(* CoDeSys 2.3.9.41 project: MO_752.pro *)
(* Libraries: STANDARD.LIB 4.10.05 11:14:46, IECSFC.LIB 13.4.06 15:51:28, SYSLIBTIME.LIB 20.2.06 13:31:16, SYSTASKINFO.LIB 20.2.06 13:31:38, ANALYZATION.LIB 5.10.99 09:05:06, arm7_specific.lib 12.5.10 15:26:52, ComService.lib 21.5.09 14:28:28, Ind_Mode.lib 26.8.10 18:05:16, ModBus.lib 27.5.09 09:22:38, Sound.lib 17.10.08 11:37:02, SysLibCom.lib 20.2.06 13:31:08, Util.lib 18.5.10 15:14:28 *)

(* PLC configuration (modules and I/O channels)
PLC73 [Root] node -1, in %IB0 out %QB0 {BName = #NМеню ПЛК73#A0; MinCycleLenght = 1; MaxCycleLenght = 1000}
  Configuration [ID10050] node 0, in %IB0 out %QB0 {BName = #NКонфигурация#A0}
    DInputs [ID10051] node 0, in %IB0.0 out %QB0.0 {BName = #NДискретные Вх.#A0}
      AT %IB0.0.0 [DInput] Битовая маска входов {CPString128 = #NСост.Дискр.Вх.#Fr.Cn#H2D26#A3#T02#O#B0120#V2; DinLM = #NЛогика Дискр.Вх#Finv.D#H62C2#A0#T02#D00#MFF#B0121#V2; DinFl = #NПост.Ф.ДребКонт#FTin.F#HF89F#A0#U0017#T02#D0A#MFF#B0122}
    Outputs [ID10057] node 1, in %IB0.1 out %QB0.1 {BName = #NВУ#A0}
      AT %QD0.1.0 [AnalogOutput0] Выход 1 {CPString128 = #NСост.ВУ1#Fr.oe#HE894#I00#A0#T00#C3#M+1.00E+00#O#B0000; AoutPWMP = #NПериод ШИМ ВУ1#Fthpd#H7BFE#I00#A0#U0017#T01#D03E8#MFDE8#L0002#B0123; AoutPWMM = #NМин.имп.ШИМ ВУ1#Ft.L#I00#B012B#A0#U0017#T01#D0032#L0001#M1388; AoutSafeValue = #NБезоп.сост.ВУ1#FO.ALr#I00#B0010#A0#C3#T00#D+0.00E+00#M+1.00E+00}
      AT %QD0.1.1 [AnalogOutput1] Выход 2 {CPString128 = #NСост.ВУ2#Fr.oe#I01#B0002#A0#O#C3#T00#M+1.00E+00; AoutPWMP = #NПериод ШИМ ВУ2#Fthpd#I01#B0124#A0#U0017#T01#D03E8#L0002#MFDE8; AoutPWMM = #NМин.имп.ШИМ ВУ2#Ft.L#I01#B012C#A0#U0017#T01#D0032#L0001#M1388; AoutSafeValue = #NБезоп.сост.ВУ2#FO.ALr#I01#B0012#A0#C3#T00#D+0.00E+00#M+1.00E+00}
      AT %QD0.1.2 [AnalogOutput2] Выход 3 {CPString128 = #NСост.ВУ3#Fr.oe#I02#B0004#A0#O#C3#T00#M+1.00E+00; AoutPWMP = #NПериод ШИМ ВУ3#Fthpd#I02#B0125#A0#U0017#T01#D03E8#L0002#MFDE8; AoutPWMM = #NМин.имп.ШИМ ВУ3#Ft.L#I02#B012D#A0#U0017#T01#D0032#L0001#M1388; AoutSafeValue = #NБезоп.сост.ВУ3#FO.ALr#I02#B0014#A0#C3#T00#D+0.00E+00#M+1.00E+00}
      AT %QD0.1.3 [AnalogOutput3] Выход 4 {CPString128 = #NСост.ВУ4#Fr.oe#HE894#I03#A0#T00#C3#M+1.00E+00#O#B0006; AoutPWMP = #NПериод ШИМ ВУ4#Fthpd#I03#B0126#A0#U0017#T01#D03E8#L0002#MFDE8; AoutPWMM = #NМин.имп.ШИМ ВУ4#Ft.L#I03#B012E#A0#U0017#T01#D0032#L0001#M1388; AoutSafeValue = #NБезоп.сост.ВУ4#FO.ALr#I03#B0016#A0#C3#T00#D+0.00E+00#M+1.00E+00}
      AT %QD0.1.4 [AnalogOutput4] Выход 5 {CPString128 = #NСост.ВУ5#Fr.oe#HE894#I04#A0#T00#C3#M+1.00E+00#O#B0008; AoutPWMP = #NПериод ШИМ ВУ5#Fthpd#I04#B0127#A0#U0017#T01#D03E8#L0002#MFDE8; AoutPWMM = #NМин.имп.ШИМ ВУ5#Ft.L#I04#B012F#A0#U0017#T01#D0032#L0001#M1388; AoutSafeValue = #NБезоп.сост.ВУ5#FO.ALr#I04#B0018#A0#C3#T00#D+0.00E+00#M+1.00E+00}
      AT %QD0.1.5 [AnalogOutput5] Выход 6 {CPString128 = #NСост.ВУ6#Fr.oe#HE894#I05#A0#T00#C3#M+1.00E+00#O#B000A; AoutPWMP = #NПериод ШИМ ВУ6#Fthpd#I05#B0128#A0#U0017#T01#D03E8#L0002#MFDE8; AoutPWMM = #NМин.имп.ШИМ ВУ6#Ft.L#I05#A0#B0130#U0017#T01#D0032#L0001#M1388; AoutSafeValue = #NБезоп.сост.ВУ6#FO.ALr#I05#B001A#A0#C3#T00#D+0.00E+00#M+1.00E+00}
      AT %QD0.1.6 [AnalogOutput6] Выход 7 {CPString128 = #NСост.ВУ7#Fr.oe#I06#B000C#A0#O#C3#T00#M+1.00E+00; AoutPWMP = #NПериод ШИМ ВУ7#Fthpd#I06#B0129#A0#U0017#T01#D03E8#L0002#MFDE8; AoutPWMM = #NМин.имп.ШИМ ВУ7#Ft.L#I06#B0131#A0#U0017#T01#D0032#L0001#M1388; AoutSafeValue = #NБезоп.сост.ВУ7#FO.ALr#I06#B001C#A0#C3#T00#D+0.00E+00#M+1.00E+00}
      AT %QD0.1.7 [AnalogOutput7] Выход 8 {CPString128 = #NСост.ВУ8#Fr.oe#I07#B000E#A0#O#C3#T00#M+1.00E+00; AoutPWMP = #NПериод ШИМ ВУ8#Fthpd#I07#B012A#A0#U0017#T01#D03E8#L0002#MFDE8; AoutPWMM = #NМин.имп.ШИМ ВУ8#Ft.L#I07#A0#B0132#U0017#T01#D0032#L0001#M1388; AoutSafeValue = #NБезоп.сост.ВУ8#FO.ALr#I07#B001E#A0#C3#T00#D+0.00E+00#M+1.00E+00}
    AInputs [ID10055] node 2, in %IB0.2 out %QB0.2 {BName = #NАналоговые Вх.#A0; Spay = #NКоррекция ХС#Fcj-.c#B0133#A0#U002A#T03#D01}
      AT %ID0.2.0 [AnalogInput0] Аналоговый вход 1 {CPString128 = #NВход 1#Fread#H8784#I00#A3#T10#C2#O#B0020#V3; AinType = #NТип датчика 1#Fin-t#H932D#I00#A0#U002F#T04#D01#M15#B0134; InFD = #NПост. фильтра 1#Fin.Fd#I00#B013C#A0#U0018#T01#D0005#M0708; InFG = #NПолоса Фильтра1#Fin.FG#I00#B0030#A0#T00#D+1.00E+01#L+0.00E+01#M+9.99E+03}
      AT %ID0.2.1 [AnalogInputTime0] Время измерения 1
      AT %ID0.2.2 [AnalogInput1] Аналоговый вход 2 {CPString128 = #NВход 2#Fread#H8784#I01#A3#T10#C2#O#B0022#V3; AinType = #NТип датчика 2#Fin-t#H932D#I01#A0#U002F#T04#D01#M15#B0135; InFD = #NПост. фильтра 2#Fin.Fd#I01#B013D#A0#U0018#T01#D0005#M0708; InFG = #NПолоса Фильтра2#Fin.FG#I01#B0032#A0#T00#D+1.00E+01#L+0.00E+01#M+9.99E+03}
      AT %ID0.2.3 [AnalogInputTime1] Время измерения 2
      AT %ID0.2.4 [AnalogInput2] Аналоговый вход 3 {CPString128 = #NВход 3#Fread#H8784#I02#A3#T10#C2#O#B0024#V3; AinType = #NТип датчика 3#Fin-t#I02#B0136#A0#U002F#T04#D01#M15; InFD = #NПост. фильтра 3#Fin.Fd#I02#B013E#A0#U0018#T01#D0005#M0708; InFG = #NПолоса Фильтра3#Fin.FG#I02#B0034#A0#T00#D+1.00E+01#L+0.00E+01#M+9.99E+03}
      AT %ID0.2.5 [AnalogInputTime2] Время измерения 3
      AT %ID0.2.6 [AnalogInput3] Аналоговый вход 4 {CPString128 = #NВход 4#Fread#H8784#I03#A3#T10#C2#O#B0026#V3; AinType = #NТип датчика 4#Fin-t#I03#B0137#A0#U002F#T04#D01#M15; InFD = #NПост. фильтра 4#Fin.Fd#I03#B013F#A0#U0018#T01#D0005#M0708; InFG = #NПолоса Фильтра4#Fin.FG#I03#A0#B0036#T00#D+1.00E+01#L+0.00E+01#M+9.99E+03}
      AT %ID0.2.7 [AnalogInputTime3] Время измерения 4
      AT %ID0.2.8 [AnalogInput4] Аналоговый вход 5 {CPString128 = #NВход 5#Fread#I04#B0028#C2#A3#O#V3#T10; AinType = #NТип датчика 5#Fin-t#I04#B0138#A0#U002F#T04#D01#M15; InFD = #NПост. фильтра 5#Fin.Fd#I04#B0140#A0#U0018#T01#D0005#M0708; InFG = #NПолоса Фильтра5#Fin.FG#I04#B0038#A0#T00#D+1.00E+01#L+0.00E+01#M+9.99E+03}
      AT %ID0.2.9 [AnalogInputTime4] Время измерения 5
      AT %ID0.2.10 [AnalogInput5] Аналоговый вход 6 {CPString128 = #NВход 6#Fread#I05#B002A#C2#A3#O#V3#T10; AinType = #NТип датчика 6#Fin-t#I05#B0139#A0#U002F#T04#D01#M15; InFD = #NПост. фильтра 6#Fin.Fd#I05#B0141#A0#U0018#T01#D0005#M0708; InFG = #NПолоса Фильтра6#Fin.FG#I05#B003A#A0#T00#D+1.00E+01#L+0.00E+01#M+9.99E+03}
      AT %ID0.2.11 [AnalogInputTime5] Время измерения 6
      AT %ID0.2.12 [AnalogInput6] Аналоговый вход 7 {CPString128 = #NВход 7#Fread#I06#B002C#C2#A3#O#V3#T10; AinType = #NТип датчика 7#Fin-t#I06#B013A#A0#U002F#T04#D01#M15; InFD = #NПост. фильтра 7#Fin.Fd#I06#B0142#A0#U0018#T01#D0005#M0708; InFG = #NПолоса Фильтра7#Fin.FG#I06#B003C#A0#T00#D+1.00E+01#L+0.00E+01#M+9.99E+03}
      AT %ID0.2.13 [AnalogInputTime6] Время измерения 7
      AT %ID0.2.14 [AnalogInput7] Аналоговый вход 8 {CPString128 = #NВход 8#Fread#H8784#I07#A3#T10#C2#O#B002E#V3; AinType = #NТип датчика 8#Fin-t#I07#B013B#A0#U002F#T04#D01#M15; InFD = #NПост. фильтра 8#Fin.Fd#I07#B0143#A0#U0018#T01#D0005#M0708; InFG = #NПолоса Фильтра8#Fin.FG#I07#B003E#A0#T00#D+1.00E+01#L+0.00E+01#M+9.99E+03}
      AT %ID0.2.15 [AnalogInputTime7] Время измерения 8
    MR1_Outputs [ID10053] node 3, in %IB0.3 out %QB0.3 {BName = #NВУ МР1#A0}
      AT %QB0.3.0 [DOutput] ВУ МР1 {CPString128 = #NСост.ВУ МР1#Fr.oe.s#HA9F4#A0#T02#O#B0144#V2}
    Additional [ID10059] node 4, in %IB0.4 out %QB0.4 {BName = #NДоп.пар-ры#A0}
      AT %QB0.4.0 [LCDLight] Подсветка {CPString128 = #NЯрк.подсв.ЖКИ#Find.i#H1845#A0#T02#D2D#M32#B0145}
      AT %QB0.4.1 [LCDContrast] Контраст {CPString128 = #NКонтраст ЖКИ#Find.C#B0146#A0#T02#D19#L05#M20}
      AT %IW0.4.2 [KBD] Клавиатура {CPString128 = #NСост.клавиатуры#Fkbrd#B0147#A3#O#T02; KBDBeep = #NЗвук кнопок#Fbeep#B0148#A0#U002A#T03#D01}
      AT %QD0.4.3 [RTS] Часы контроллера {RTSPar = #NВремя и дата#FrtC#HFA30#A0#T05#O#B0040}
      AT %QB0.4.4 [LED] Светодиоды {CPString128 = #NСос.светодиодов#Find.L#HF304#A0#T02#D00#M3F#L00#O#B0149#V2}
    Versions [ID10060] node 5, in %IB0.5 out %QB0.5 {BName = #NВерсииПрошивок#A0}
      AT %QB0.5.0 [DevName] Имя устройства {CPString128 = #NИмя устройства#Fdev#B0042#A3#O#T08}
      AT %IB0.5.1 [HardVer] Прошивка {CPString128 = #NВерсия прошивки#Fver#B004A#A3#O#T08}
      AT %QB0.5.2 [SoftVer] Программа {CPString128 = #NВерсияПрограммы#Fp.ver#B0052#A3#O#T08}
    RS-1 [ID10061] node 6, in %IB0.6 out %QB0.6 {BName = #NНастр.RS-1#A0; RSBPS = #NСкорость#FbPS#I00#B014A#A0#U0046#T04#D00#M09; RSWLen = #NДлина слова#FLen#I00#B014B#A0#U0005#T04#D03#M03; RSPrt = #NЧётность#Fprty#I00#B014C#A0#U009A#T04#D04#M04; RSStp = #NСтоп биты#Fsbit#I00#B014D#A0#U00A1#T04#D00#M02; RSALen = #NДлина адреса#Fa.len#I00#B014E#A0#U0055#T03#D00; RSAdr = #NАдрес прибора#FAddr#I00#B014F#A0#T01#D0010#M07FF; RSDl = #NЗадержка ответа#FRs.dl#I00#B0150#A0#U0017#T02#D05#M32}
    RS-2 [ID10062] node 7, in %IB0.7 out %QB0.7 {BName = #NНастр.RS-2#A0; RSBPS = #NСкорость#FbPS#I01#B0151#A0#U0046#T04#D00#M09; RSWLen = #NДлина слова#FLen#I01#B0152#A0#U0005#T04#D03#M03; RSPrt = #NЧётность#Fprty#I01#B0153#A0#U009A#T04#D04#M04; RSStp = #NСтоп биты#Fsbit#I01#B0154#A0#U00A1#T04#D00#M02; RSALen = #NДлина адреса#Fa.len#I01#B0155#A0#U0055#T03#D00; RSAdr = #NАдрес прибора#FAddr#I01#B0156#A0#T01#D0010#M07FF; RSDl = #NЗадержка ответа#FRs.dl#I01#B0157#A0#U0017#T02#D05#M32}
  WorkInd [ID10100] node 1, in %IB1 out %QB1 {WIChanelCount = 6}
  SubMenu [ID11000] node 2, in %IB2 out %QB2 {BName = #NВетка#A0}
  SubMenu [ID11000] node 3, in %IB3 out %QB3 {BName = #NВетка#A0}
  SubMenu [ID11000] node 4, in %IB4 out %QB4 {BName = #NВетка#A0}
*)

(* Global variable list: Global_Variables *)
VAR_GLOBAL CONSTANT

	byMU110Address: BYTE:=11;				(*адрес МУ-110*)
	byMV110Address: BYTE:=22;				(*адрес МВ-110*)

END_VAR
VAR_GLOBAL
	bDInput1 AT %IX0.0.0.0: BOOL;
	bDInput2 AT %IX0.0.0.1: BOOL;
	bDInput3 AT %IX0.0.0.2: BOOL;
	bDInput4 AT %IX0.0.0.3: BOOL;
	bDInput5 AT %IX0.0.0.4: BOOL;
	bDInput6 AT %IX0.0.0.5: BOOL;
	bDInput7 AT %IX0.0.0.6: BOOL;
	bDInput8 AT %IX0.0.0.7: BOOL;

	rOutput1 AT %QD0.1.0: REAL;
	rOutput2 AT %QD0.1.1: REAL;
	rOutput3 AT %QD0.1.2: REAL;
	rOutput4 AT %QD0.1.3: REAL;
	rOutput5 AT %QD0.1.4: REAL;
	rOutput6 AT %QD0.1.5: REAL;
	rOutput7 AT %QD0.1.6: REAL;
	rOutput8 AT %QD0.1.7: REAL;

	rAInput1 AT %ID0.2.0: REAL;
	rAInput2 AT %ID0.2.2: REAL;
	rAInput3 AT %ID0.2.4: REAL;
	rAInput4 AT %ID0.2.6: REAL;
	rAInput5 AT %ID0.2.8: REAL;
	rAInput6 AT %ID0.2.10: REAL;
	rAInput7 AT %ID0.2.12: REAL;
	rAInput8 AT %ID0.2.14: REAL;

	kbrd AT %IW0.4.2: WORD;
	led  AT %QB0.4.4: BYTE;
	n: WORD := 0;
END_VAR
VAR_GLOBAL RETAIN
	wFilterTimeRet: 	WORD	:= 3000;    (*время фильтра поплавка в мс*)
	tempMaxRet: 		BYTE	:= 95;		(*максим. температура*)
	timeMaxRet: 		WORD	:= 999;		(*максим. время*)
	USDelayRet: 		WORD	:= 0;		(*время блокировки повторного включения УЗ в сек*)
	hystRet: 			WORD	:= 2;		(*гистерезис *10^(-2) гр.С*)
	pumpModeRet: 	    BOOL;				(*режим работы насоса (TRUE - работает постоянно, FALSE - с заданной частотой и скважностью*)
	pumpTimeLo:         WORD;				(*массив для задания времени бездействия насоса в минутах*)
	pumpTimeHi: 		WORD;				(*массив для задания продолжительности работы насоса в секундах*)
	APRet: 		        ARRAY [US_1..Wash] OF APST;				(*параметры автоматической программы*)
	powerOffDelayRet: 	WORD	:= 15;		(*задержка отключения питания генераторов в секундах*)
	genOnDelayRet: 	    WORD	:= 500;		(*время между включениями генераторов в мс*)
    fillDelay:          WORD    := 5;       (*задержка закрытия электроклапана наполнения воды*)
    ventTime:           WORD    := 0;       (*задержка гидролока*)
	timePump:			WORD    := 1;
	temp_Air:			WORD;
	time_dry:			WORD;
END_VAR

(* Global variable list: GVL_APBool *)
VAR_GLOBAL CONSTANT
    WarmWait :BYTE:=0;    (*отложенный старт*)
    DynContr :BYTE:=1;    (*динамическое управление*)
    RotOn    :BYTE:=2;    (*качание*)
END_VAR

(* Global variable list: GVL_CONST *)
VAR_GLOBAL CONSTANT
	iQtyD7Line: 		INT		:=25;		(*количество строк в расписании недельного таймера*)
	iMaxSelScrParam: 	INT		:=26;		(*максимальное количество строк на экране выбора параметра*)
	iStQty: 			INT		:=10;		(*количество шагов автоматической программы*)
	tUSDelay: 			TIME	:=t#1m;		(*задержка повторной подачи питания на УЗГ*)
	GlobalMaxRand: 		USINT	:=18;		(*количество рандомных значений и максимальное значение рандома*)
END_VAR

(* Data type in BathFB *)
TYPE APST :
STRUCT
	areSt:		ARRAY [1..iStQty] OF StAPE;        (*массив шагов автоматической программы*)
	arwTime:	ARRAY [1..iStQty] OF WORD;         (*временной параметр шага в минутах*)
	byTemp:		BYTE;                              (*заданная температура*)
	byBool:		BYTE;                              (*состояние программных ключей. Описываются в GVL_APBoolE*)
	byTempAir:	BYTE;
END_STRUCT
END_TYPE

(* Data type *)
TYPE Button :
STRUCT
    pusk:            ARRAY [US_1..Wash] OF BOOL;   (*Пуск*)
    stop:            ARRAY [US_1..Wash] OF BOOL;   (*Стоп*)
    emStop:          BOOL;   (*Аварийный стоп*)
	pusk_dry:		BOOL;
	stop_dry:		BOOL;
    puskDrain:       BOOL;   (*Пуск слива*)
    puskFill:        BOOL;   (*Пуск наполнения*)
    puskPump:        BOOL;   (*Пуск насоса*)
    puskBubbles:     BOOL;   (*Пуск барботажа*)
	warmOn:          BOOL;
END_STRUCT
END_TYPE

(* Data type in BathFB *)
TYPE ButtonBath :
STRUCT
	Pusk:          BOOL;   (*Пуск цикла*)
	PuskDrain:     BOOL;   (*Пуск слива*)
	PuskFill:      BOOL;   (*Пуск наполнения*)
	PuskPump:      BOOL;   (*Пуск насоса*)
	PuskBubbles:   BOOL;   (*Пуск барботажа*)
	Stop:          BOOL;   (*Стоп*)
	StopDrain:     BOOL;   (*Стоп слива*)
	StopFill:      BOOL;   (*Стоп наполнения*)
	emStop:        BOOL;   (*Аварийная остановка*)
END_STRUCT
END_TYPE

(* Data type in BathFB *)
TYPE ButtonEvent :
STRUCT
   (* кнопка нажата, устанавливается на один цикл *)
   downEvent:    BOOL;

   (* нажатие дольше секунды *)
   longPush:     BOOL;

   (* число, на которое надо инкрементировать, сначала 1,
   начиная с 3 секунды увеличиваеться на 1 каждую секунду *) 
   incr:         BYTE;
END_STRUCT
END_TYPE

(* Data type *)
TYPE Control :
STRUCT
	heatUSTank:		BOOL;                    (*нагрев в баке УЗВ*)
	heatWashTank:	BOOL;                    (*нагрев в баке ополаскивания*)
	pump:			BOOL;                    (*насосы*)
	lampAtt:		BOOL;                    (*лампа "Внимание"*)
	warning_bath:	ARRAY [US_1..Wash] OF BOOL;
	warning_dry:	BOOL;
	lampWork:		BOOL;                    (*лампа "Работа"*)
	lamp_work_dry:	BOOL;
	lamp_work_bath:	ARRAY [US_1..US_2] OF BOOL;
	lampTopLevel:	BOOL;                    (*лампа "Верхняя группа УЗГ"*)
	lampLowerLevel:	BOOL;                    (*лампа "Нижняя группа УЗГ"*)
	genPower:		BOOL;                    (*питание генераторов*)
	skim:			BOOL;                    (*скиммеры*)
	gener:			ARRAY [1..36] OF BOOL;   (*генераторы*)
	heat_air:		BOOL;
	fan:			BOOL;
END_STRUCT
END_TYPE

(* Data type in BathFB *)
TYPE ControlBath :
STRUCT
   us:                  BOOL;      (*ультразвук*)
   warmBath:            BOOL;      (*нагрев ванны*)
   warmTank:            BOOL;      (*нагрев бака*)
   rotFo:               BOOL;      (*вращение вперед*)
   rotRe:               BOOL;      (*вращение назад*)
   ventBfromNet:        BOOL;      (*вентиль из сети*)
   pumpBfromTank:       BOOL;      (*фильтрационный насос*)
   ventBPocketToNet:    BOOL;      (*вентиль из кармана в сеть*)
   ventBPocketToTank:   BOOL;      (*вентиль из кармана в бак*)
   ventBToNet:          BOOL;      (*вентиль из ванны в сеть*)
   ventBToTank:         BOOL;      (*вентиль из ванны в бак*)
   ventBarb:            BOOL;      (*барботаж*)
   skim:                BOOL;      (*скиммер*)
   dry:                 BOOL;      (*сушка*)
   dryFan:              BOOL;      (*вентилятор сушки*)
END_STRUCT
END_TYPE

(* Data type in D7Timer *)
TYPE D7TLineST :    (*структура одной линии расписания 7дн таймера*)
STRUCT
    wTimeOfWeek:    WORD;    (*время недели в минутах, к этому времени надо нагреть*)
    byTemp:         BYTE;    (*поддерживаемая температура*)
    byDur:          BYTE;    (*продолжительность в часах*)
END_STRUCT
END_TYPE

(* Data type in D7Timer *)
TYPE DoWE :
(
    Mon:=0,
    Tue,
    Wed,
    Thu,
    Fri,
    Sat,
    Sun
);
END_TYPE

(* Data type in BathFB *)
(*Дополнительные выходы ванны*)
TYPE ExtOutST :
STRUCT
    remTime:     TIME;    (*оставшееся время*)
    bathEmpty:   BOOL;    (*ванна пуста*)
END_STRUCT
END_TYPE

(* Data type in BathFB *)
(*дополнительные параметры ванны*)
TYPE ExtParamST :
STRUCT
    (*Нагреватели*)
    heatPlace:        HeatPlaceE;    (*место расположения нагревателя*)
    heaterInTank:     BOOL;          (*расположение ТЭН в баке*)
    deltaHyst:        WORD;          (*гистерезис нагрева (e(-2))*)
    waitTemp:         BYTE;          (*температура режима ожидания (с недельного таймера или заданная вручную)*)
    mixTimeHi:        WORD;          (*время работы перемешивания в секундах*)
    mixTimeLo:        WORD;          (*время ожидания перемешивания в минутах*)
    pumpTimeHi:       WORD;          (*работа насоса в секундах*)
    pumpTimeLo:       WORD;          (*ожидание насоса в минутах*)
    mixStart:         BOOL;          (*время между включениями барботажа при нагреве в минутах*)
    mixDur:           WORD;          (*время барботажа при нагреве в секундах*)

    (*Вентили*)
    ventTime:         WORD;          (*время работы вентиля в секундах*)
    drainDelay:       WORD;          (*дополнительное время слива в секундах*)
    fillDelay:        WORD;          (*дополнтельное время наполнения в секундах*)
    pumpDelay:        WORD;          (*дополнительное время насоса в секундах*)
    fillTankDelay:    WORD;          (*дополнительное время наполнения бака в секундах*)
    dontDrain:        BOOL;          (*не сливать ванну*)

    (*барабан*)
    rotTime:          WORD;          (*период качания в миллисекундах*)
    rotDur:           WORD;          (*продолжительность качания в секундах*)
    rotSlack:         WORD;          (*продолжительность бездействия в секундах*)
    filtrRot:         BOOL;          (*вращение при фильтрации*)

    (*скиммер*)
    skimTimeHi:       WORD;          (*время работы скиммера в минутах*)
    skimTimeLo:       WORD;          (*время ожидания скиммера в минутах*)

END_STRUCT
END_TYPE

(* Data type in BathFB *)
TYPE FlE :
(
    NoFl,    (*нет жидкости*)
    TMS,
    water
);
END_TYPE

(* Data type in BathFB *)
(*расположение нагревателя*)
TYPE HeatPlaceE :
(
    US_1,
    US_2,
    Wash
);
END_TYPE

(* Data type in Other *)
TYPE kbrd_tip :
(
    off:=0,
    DOWN:=4,
    UP:=8,
    ENTER:=16,
    OUT:=64,
    ALT:=128,
    F1:=1,
    F2:=2,
    F3:=256,
    pusk_stop:=32,
    ALT_F1:=129,
    ALT_F3:=384
);
END_TYPE

(* Data type *)
TYPE Level :
(
    BathTop,
    BathMiddle,
    BathLower,
    TankTop,
    TankMiddle,
    TankLower,
    USBlock,
    USBlockTop,
    WarmBlock,
    PumpBlock,
    BarbBlock,
    SkimerBlock,
    FillBathStop
);
END_TYPE

(* Data type in BathFB *)
TYPE LevelBath :
STRUCT
    BathTop:        BOOL;       (*Верхний уровень в ванне*)
    BathMiddle:     BOOL;       (*Средний уровень в ванне*)
    BathLower:      BOOL;       (*Нижний уровень в ванне*)
    TankTop:        BOOL;       (*Верхний уровень в баке*)
    TankMiddle:     BOOL;       (*Средний уровень в баке*)
    TankLower:      BOOL;       (*Нижний уровень в баке*)
    USBlock:        BOOL;       (*Уровень блокировки уровня ультразвука*)
    USBlockTop:     BOOL;       (*Уровень блокировки верхнего уровня ультразвука*)
    WarmBlock:      BOOL;       (*Уровень блокировки нагрева*)
    PumpBlock:      BOOL;       (*Уровень блокировки насоса*)
    BarbBlock:      BOOL;       (*Уровень блокировки барботажа*)
    SkimerBlock:    BOOL;       (*Уровень блокировки скимера*)
    FillBathStop:   BOOL;       (*Уровень заполнения*)
END_STRUCT
END_TYPE

(* Data type *)
TYPE MBStepE :
(
    StepSelect,
    MV110Read,
    MU110Write
);
END_TYPE

(* Data type *)
TYPE ModuleAddr :
(
    A2 := 22,
    A3 := 33,
    A4 := 44,
    A5 := 55,
    A6 := 66,
    A7 := 77
);
END_TYPE

(* Data type *)
TYPE Screens :
(
	s_info,

	s_osnovnoy_US_1,
	s_osnovnoy_US_2,
	s_osnovnoy_Wash,
	s_osnovnoy_Dry,

	s_nastroyki,
	s_nastroyki_ext,

	s_time,
	s_time_us_1,
	s_time_us_2,
	s_time_dry,

	s_tem,
	s_tem_us_1,
	s_tem_us_2,
	s_tem_wash,
	s_tem_dry,

	s_tMaxSet,
	s_temHSet
);
END_TYPE

(* Data type in Other *)
TYPE SelectScreenAddStruc :
STRUCT
    strIn: STRING(5);    (*строка, дописываемая между ВЫХОД и ВХОД*)
END_STRUCT
END_TYPE

(* Data type *)
TYPE Sensor :
STRUCT
    level:			ARRAY [BathTop..FillBathStop, US_1..Wash] OF BOOL;	(*массив уровней*)
    button:			Button;									(*кнопки*)
    genState:		ARRAY [1..36] OF BOOL;					(*состояние генераторов*)
    tempBath:		ARRAY [US_1..Wash] OF REAL;				(*температура ванны*)
    overloadPump:	BOOL;									(*Перегрев насоса*)
	temAir:			REAL;
	cover:			BOOL;
END_STRUCT
END_TYPE

(* Data type in BathFB *)
TYPE SensorBath :
STRUCT
    level:			LevelBath;   (*Уровни*)
    tempBath:		REAL;        (*Температура ванны*)
    tempTank:		REAL;        (*Температура бака*)
	tempAir:		REAL;
	button:			ButtonBath;  (*Кнопки*)
    Fl:				FlE;         (*тип жидкости в ванне*)
    warmOn:			BOOL;        (*нагрев включен*)
    mixOn:			BOOL;        (*перемешивание включен*)
    pause:			BOOL;        (*Пауза АП*)
    rotOn:			BOOL;        (*Включение вращения*)
    flReset:		BOOL;        (*Сброс типа жидкости*)
	overloadPump:	BOOL;        (*перегрузка насоса*)
END_STRUCT
END_TYPE

(* Data type in Other *)
(*дополнительные настройки для блока экрана установки параметра*)
TYPE SetScreenAddStruc :
STRUCT
    Extend:        BOOL;                        (*разрешает работу блока в режиме задания разных велечин*)
    in_var:        ARRAY[1..3] OF DWORD;        (*задаваемая переменная*)
    in_var_min:    ARRAY[1..3] OF  DWORD;       (*мин значение задаваемой переменной*)
    in_var_max:    ARRAY[1..3] OF  DWORD;       (*макс значение задаваемой переменной*)
    UnitParam:     ARRAY[1..3] OF  STRING(16);  (*в каких единицах ведется задание минуты секунды градусы и тд*)
    EnableF3:      BOOL;                        (*разрешить третью единицу измерения*)
    bDoWSet:       BOOL;                        (*задаваемый параметр - день недели*)
    iValInc:       INT;                         (*шаг увеличения величины*)
END_STRUCT
END_TYPE

(* Data type in Other *)
TYPE StAPE:
(
    Wait:=0,
    WarmTank,
    WarmBath,
    FillFromTank,
    US,
    FiltrToTank,
    DrainToTank,
    FillFromNet,
    US2,
    FiltrToNet,
    DrainToNet,
    FillTank,
    ManToNet,
    ManToTank,
    Skip,
    Barb,
    Barb_and_Filtr,
    Dry,
    DeGas,
    Warning,
    Pump,
	Cooling,
	Heating
);
END_TYPE

(* Data type in BathFB *)
TYPE StE :
(
    on,
    off1,
    not_enabled
);
END_TYPE

(* Data type *)
TYPE VarST :
STRUCT
    pby:      POINTER TO BYTE;
    type_:    VarType;
END_STRUCT
END_TYPE

(* Data type *)
TYPE VarType :
(
    BYTE_,
    WORD_,
    DWORD_,
    REAL_,
    DINT_,
    DWORD_30,
    DWORD_500
);
END_TYPE

(* POU PLC_PRG, ST *)
PROGRAM PLC_PRG
VAR
	bInit:              BOOL;
	warning:            BOOL;
	C:                  INT;
	D:                  BOOL;

	encoder_:			Encoder;
	TON50ms:            TON;

	bath:               ARRAY [US_1..Wash] OF BFBv4;                           (*массив ФБ ванн*)
	block:              ARRAY [US_1..Wash] OF BlockFBv2;                       (*блокировки*)
	sens:               Sensor;                          (*структура датчиков*)
	contr:              Control;                         (*структура управления*)
	filtr:              digitalFiltr;
	buttons:            KeyboardFB;
	variable:           VarST;
	HYST_Air:			HYST;
	TON_heat_air:		TON;
	TON_fan:			TON;
	TONP:				TONP;
	start_heat_air:		BOOL;
	stape:				StAPE;

	(*modbus*)
	bOpenPort:          BOOL        := 0;
	ePorts:             PORTS       := 0;
	stSettings:         COMSETTINGS;
	oComService:        COM_SERVICE;
	arMBuffer:          ARRAY [0..255] OF BYTE;
	tTimeOut:           TIME        := t#100ms;      (*время таймаута порта*)
	eMBStep:            MBStepE     := MV110Read;  (*кейс модбаса*)
	udErr:              UDINT       :=0;            (*счетчик ошибок*)
	wBuffer:            WORD;

	mbA2:               WORD;
	arTON:              ARRAY [1..2] OF TON;

	oMB_16:             MB_WR_REGS;                 (*функция Modbus 16*)
	oMB_03:             MB_RD_HOLD_REGS;            (*функция Modbus 03*)
	oMB_06:				MB_WR_SNG_REG;				(*запись значения в один регистр хранения (Preset Single Register).*)

	TONMBDelay:         TON;                        (*таймер задержки modbus*)
	tMBDelay:           TIME        := t#10ms;     (*задержка modbus*)
	bMBStepSelect:      BOOL;                       (*выбор запись/чтение*)

	(*indicator*)
	Current_screen:     screens     := s_info;
	TONInfo:            TON;
	str:                ARRAY [1..4] OF STRING(16);
	pred_str:           ARRAY [1..4] OF STRING(16);
	SelectScreen:       SelectScreenFB;
	SetScreen:          SetScreenFB;

END_VAR
VAR_TEMP

	I:                  INT;
	k:                  INT;
	j:                  INT;
	iStTmp:             INT;                        (*шаг АП*)
	line:               INT;                        (*строка индикатора*)

END_VAR
IF NOT(bInit) THEN
    acInit();									(*инициализация*)
ELSE

	buttons(kbrd := kbrd);
	acMB();
	SelectScreen.encoder_(A := bDInput6, B := bDInput5, button := bDInput7, connected := TRUE);
	SetScreen.pSelect := ADR(SelectScreen);
	C := SelectScreen.encoder_.counter;
	D := SelectScreen.encoder_.press;

	encoder_(A := bDInput6, B := bDInput5, button := bDInput7, connected := TRUE);


	(*назначение входов*)
	sens.tempBath[US_1]			:= rAInput1;
	sens.tempBath[US_2]			:= rAInput2;
	sens.tempBath[Wash]			:= rAInput3;
	sens.temAir					:= rAInput4;

	sens.button.emStop			:= bDInput1;

	sens.level[BathLower, US_1]	:= mbA2.0;
	sens.level[BathLower, US_2]	:= mbA2.1;
	sens.level[BathLower, Wash]	:= mbA2.2;
	sens.button.pusk[US_1]		:= mbA2.4;
	sens.button.stop[US_1]		:= mbA2.5;
	sens.button.pusk[US_2]		:= mbA2.6;
	sens.button.stop[US_2]		:= mbA2.7;
	sens.button.pusk_dry		:= mbA2.8;
	(*sens.button.stop_dry		:= mbA2.9;*)

	(*назначение входов ванн*)
	FOR i := US_1 TO Wash DO
		bath[i].sens.button.Pusk               := sens.button.pusk[i];
		bath[i].sens.button.Stop               := sens.button.stop[i] ;
		bath[i].sens.pause                     := NOT sens.level[BathLower, i];
		bath[i].sens.tempBath                  := sens.tempBath[i];
		bath[i].sens.level.BathLower           := sens.level[BathLower, i];
		bath[i].sens.warmOn                    := TRUE;
		bath[i].param.heaterInTank             := TRUE;
		bath[i].param.deltaHyst                := hystRet;
		bath[i].sens.button.emStop             := sens.button.emStop;
		bath[i].sens.level.USBlock := bath[i].sens.level.WarmBlock := bath[i].sens.level.BathLower;
	END_FOR


	FOR i := US_1 TO Wash DO
		bath[i](stAP:=APRet[i]);
		block[i]();
	END_FOR

	(*управление*)
	CASE stape OF
		Wait:
			contr.heat_air	:= FALSE;
			contr.fan		:= FALSE;
			IF sens.button.pusk_dry AND (temp_Air <> 0) AND (time_dry <> 0) THEN
				stape := Heating;
			END_IF
		Heating:
			contr.heat_air := HYST_Air.nagrev;
			contr.fan := TRUE;
			IF sens.temAir >= temp_Air THEN
				stape:= Dry;
			END_IF
			IF sens.button.stop_dry THEN
				contr.heat_air := FALSE;
				stape := Cooling;
			END_IF
		Dry:
			contr.heat_air := HYST_Air.nagrev;
			contr.fan := TRUE;
			TONP(P := FALSE, IN := TRUE, PT := TO_MIN(time_dry));
			IF TONP.Q OR sens.button.stop_dry THEN
				contr.heat_air := FALSE;
				TONP(IN:= FALSE);
				stape := Cooling;
			END_IF
		Cooling:
			TON_fan(IN := TRUE, PT := TO_MIN(5));
			IF TON_fan.Q THEN
				TON_fan(IN:= FALSE);
				stape := Wait;
			END_IF
	END_CASE

	HYST_Air.temperatura := temp_Air;
	HYST_Air(ENABLE := stape = Dry OR stape = Heating, temInput := sens.temAir	, temperaturaH := hystRet);

	FOR i := US_1 TO Wash DO
		contr.warning_bath[i]	:= NOT bath[i].sens.level.BathLower OR bath[i].sens.button.emStop OR (bath[i].sens.tempBath < 0);
	END_FOR
	contr.warning_dry			:= sens.temAir < 0;



	contr.lamp_work_bath[US_1]	:= bath[US_1].eStAP <> Wait;
	contr.lamp_work_bath[US_2]	:= bath[US_2].eStAP <> Wait;
	contr.lamp_work_dry			:= stape <> Wait;
	contr.lampAtt				:= contr.warning_bath[US_1] OR contr.warning_bath[US_2] OR contr.warning_bath[Wash] OR contr.warning_dry;

	(*Назначение выходов*)
	rOutput3 := BOOL_TO_REAL(contr.lampAtt);
	rOutput1 := BOOL_TO_REAL(contr.lamp_work_bath[US_1] OR contr.lamp_work_bath[US_2] OR contr.lamp_work_dry);

	rOutput5 := BOOL_TO_REAL(contr.lamp_work_bath[US_1]);
	rOutput6 := BOOL_TO_REAL(contr.lamp_work_bath[US_2]);
	rOutput7 := BOOL_TO_REAL(contr.lamp_work_dry);

	led.0 := contr.warning_bath[US_1];
	led.1 := contr.warning_bath[US_2];
	led.2 := contr.warning_bath[Wash];
	led.3 := contr.warning_dry;

	(*вызов действия индикации*)
	TON50ms(IN:=TRUE,PT:=t#50ms);
	IF TON50ms.Q THEN
		TON50ms(IN:=FALSE);
		acIndicator();
	END_IF
END_IF
END_PROGRAM
ACTION acIndicator:
CASE Current_screen OF

	s_info:

		Switch_To_Single_Mode();				(*переход в монопольный режим*)
		str[1] := '      ООО       ';
		str[2] := 'Александра-Плюс ';
		str[3] := '                ';
		str[4] := '     МО-752     ';
		TONInfo(IN := TRUE, PT := t#5s);
		IF TONInfo.Q THEN
			TONInfo(IN := FALSE);
			encoder_(reset := TRUE);
			Current_screen := s_osnovnoy_US_1;
		END_IF

	s_osnovnoy_US_1:
		encoder_(reset := FALSE);
		SelectScreen(kbrd := kbrd, QtyParam := 3);
		line := 1;
		str[line] := ' МО-752    УЗВ1 ';
		line := 2;
		IF bath[US_1].eStAP <> Wait THEN
			str[line] := CONCAT('Время     ', TIME_TO_MMSS(bath[US_1].extOutB.remTime));
		ELSE
			str[line] := CONCAT('Время     ', TIME_TO_MMSS(TO_MIN(APRet[US_1].arwTime[2])));
		END_IF

		line := 3;
		str[line] := CONCAT('Нагрев ', TEMP_TO_STRING(bath[US_1].sens.tempBath));
		str[line] := CONCAT(str[line], '/');
		str[line] := CONCAT(str[line], DWORD_TO_STRING (APRet[US_1].byTemp ));
		str[line] := CONCAT(str[line], '$9BС');
		line := 4;
		IF sens.tempBath[US_1] < 0 THEN
			str[line] := ' неисправно ТС  ';
			warning :=TRUE;
		ELSIF sens.button.emStop  THEN
			str[line] := ' Авар. останов! ';
			warning :=TRUE;
		ELSIF NOT bath[US_1].sens.level.BathLower  THEN
			str[line] := 'низкий ур. р-ра ';
			warning :=TRUE;
		ELSIF stape = Heating THEN
			str[line] := '    подогрев    ';
			warning :=FALSE;
		ELSIF stape = Dry THEN
			str[line] := '     сушка      ';
			warning :=FALSE;
		ELSIF bath[US_1].eStAP = US THEN
			str[line] := '   ультразвук   ';
			warning :=FALSE;
		ELSIF stape = Cooling THEN
			str[line] := '   охлаждение   ';
			warning :=FALSE;
		ELSIF bath[US_1].eStAP = Wait THEN
			str[line] := 'ожидание старта ';
			warning :=FALSE;
		END_IF
		IF SelectScreen.encoder_.press AND SelectScreen.encoder_.enable OR SelectScreen.kbrd = F1 THEN
			SelectScreen.encoder_(enable := FALSE);
			Current_screen := s_nastroyki;
		END_IF
		IF SelectScreen.kbrd = ALT_F3 THEN
			Current_screen := s_nastroyki_ext;
		END_IF

		IF (encoder_.counter >= 1) THEN
			Current_screen := s_osnovnoy_US_2;
			encoder_(reset := TRUE);
		ELSIF encoder_.counter < 0 THEN
			encoder_(reset := TRUE);
		END_IF


	s_osnovnoy_US_2:
		encoder_(reset := FALSE);
		SelectScreen(kbrd := kbrd, QtyParam := 3);
		line := 1;
		str[line] := ' МО-752    УЗВ2 ';
		line := 2;
		IF bath[US_2].eStAP <> Wait THEN
			str[line] := CONCAT('Время     ', TIME_TO_MMSS(bath[US_2].extOutB.remTime));
		ELSE
			str[line] := CONCAT('Время     ', TIME_TO_MMSS(TO_MIN(APRet[US_2].arwTime[2])));
		END_IF

		line := 3;
		str[line] := CONCAT('Нагрев ', TEMP_TO_STRING(bath[US_2].sens.tempBath));
		str[line] := CONCAT(str[line], '/');
		str[line] := CONCAT(str[line], DWORD_TO_STRING (APRet[US_2].byTemp ));
		str[line] := CONCAT(str[line], '$9BС');
		line := 4;
		IF sens.tempBath[US_2] < 0 THEN
			str[line] := ' неисправно ТС  ';
			warning :=TRUE;
		ELSIF sens.button.emStop  THEN
			str[line] := ' Авар. останов! ';
			warning :=TRUE;
		ELSIF NOT bath[US_2].sens.level.BathLower  THEN
			str[line] := 'низкий ур. р-ра ';
			warning :=TRUE;
		ELSIF stape = Heating THEN
			str[line] := '    подогрев    ';
			warning :=FALSE;
		ELSIF stape = Dry THEN
			str[line] := '     сушка      ';
			warning :=FALSE;
		ELSIF bath[US_2].eStAP = US THEN
			str[line] := '   ультразвук   ';
			warning :=FALSE;
		ELSIF stape = Cooling THEN
			str[line] := '   охлаждение   ';
			warning :=FALSE;
		ELSIF bath[US_2].eStAP = Wait THEN
			str[line] := 'ожидание старта ';
			warning :=FALSE;
		END_IF
		IF SelectScreen.encoder_.press AND SelectScreen.encoder_.enable OR SelectScreen.kbrd = F1 THEN
			SelectScreen.encoder_(enable := FALSE);
			Current_screen := s_nastroyki;
		END_IF
		IF SelectScreen.kbrd = ALT_F3 THEN
			Current_screen := s_nastroyki_ext;
		END_IF
		IF (encoder_.counter <= - 1) THEN
			Current_screen := s_osnovnoy_US_1;
			encoder_(reset := TRUE);
		ELSIF (encoder_.counter >= 1) THEN
			Current_screen := s_osnovnoy_Wash;
			encoder_(reset := TRUE);
		END_IF

	s_osnovnoy_Wash:
		encoder_(reset := FALSE);
		SelectScreen(kbrd := kbrd, QtyParam := 3);
		line := 1;
		str[line] := ' МО-752 ополаск.';
		line := 2;
		str[line] := '                ';
		line := 3;
		str[line] := CONCAT('Нагрев ', TEMP_TO_STRING(bath[Wash].sens.tempBath));
		str[line] := CONCAT(str[line], '/');
		str[line] := CONCAT(str[line], DWORD_TO_STRING (APRet[Wash].byTemp ));
		str[line] := CONCAT(str[line], '$9BС');
		line := 4;
		IF sens.tempBath[Wash] < 0 THEN
			str[line] := ' неисправно ТС  ';
			warning :=TRUE;
		ELSIF sens.button.emStop  THEN
			str[line] := ' Авар. останов! ';
			warning :=TRUE;
		ELSIF NOT bath[Wash].sens.level.BathLower  THEN
			str[line] := 'низкий ур. р-ра ';
			warning :=TRUE;
		ELSIF stape = Heating THEN
			str[line] := '    подогрев    ';
			warning :=FALSE;
		ELSIF stape = Dry THEN
			str[line] := '     сушка      ';
			warning :=FALSE;
		ELSIF stape = Cooling THEN
			str[line] := '   охлаждение   ';
			warning :=FALSE;
		ELSIF bath[Wash].eStAP = Wait THEN
			str[line] := '                ';
			warning :=FALSE;
		END_IF
		IF SelectScreen.encoder_.press AND SelectScreen.encoder_.enable OR SelectScreen.kbrd = F1 THEN
			SelectScreen.encoder_(enable := FALSE);
			Current_screen := s_nastroyki;
		END_IF
		IF SelectScreen.kbrd = ALT_F3 THEN
			Current_screen := s_nastroyki_ext;
		END_IF

		IF (encoder_.counter <= - 1) THEN
			Current_screen := s_osnovnoy_US_2;
			encoder_(reset := TRUE);
		ELSIF (encoder_.counter >= 1) THEN
			Current_screen := s_osnovnoy_Dry;
			encoder_(reset := TRUE);
		END_IF


	s_osnovnoy_Dry:
		encoder_(reset := FALSE);
		SelectScreen(kbrd := kbrd, QtyParam := 3);
		line := 1;
		str[line] := ' МО-752   Сушка ';
		line := 2;
		IF stape = Dry THEN
			str[line] := CONCAT('Время     ', TIME_TO_MMSS(TO_MIN(time_dry) - TONP.ET));
		ELSIF stape = Cooling THEN
			str[line] := CONCAT('Время     ', TIME_TO_MMSS(TO_MIN(5) - TON_fan.ET));
		ELSE
			str[line] := CONCAT('Время     ', TIME_TO_MMSS(TO_MIN(time_dry)));
		END_IF

		line := 3;
		str[line] := CONCAT('Нагрев ', TEMP_TO_STRING(sens.temAir));
		str[line] := CONCAT(str[line], '/');
		str[line] := CONCAT(str[line], DWORD_TO_STRING (temp_Air ));
		str[line] := CONCAT(str[line], '$9BС');
		line := 4;
		IF sens.temAir < 0 THEN
			str[line] := ' неисправно ТС  ';
			warning :=TRUE;
		ELSIF sens.button.emStop  THEN
			str[line] := ' Авар. останов! ';
			warning :=TRUE;
		ELSIF stape = Heating THEN
			str[line] := '    подогрев    ';
			warning :=FALSE;
		ELSIF stape = Dry THEN
			str[line] := '     сушка      ';
			warning :=FALSE;
		ELSIF stape = Cooling THEN
			str[line] := '   охлаждение   ';
			warning :=FALSE;
		ELSIF stape = Wait THEN
			str[line] := 'ожидание старта ';
			warning :=FALSE;
		END_IF

		IF SelectScreen.encoder_.press AND SelectScreen.encoder_.enable OR SelectScreen.kbrd = F1 THEN
			SelectScreen.encoder_(enable := FALSE);
			Current_screen := s_nastroyki;
		END_IF

		IF SelectScreen.kbrd = ALT_F3 THEN
			Current_screen := s_nastroyki_ext;
		END_IF

		IF (encoder_.counter <= - 1) THEN
			Current_screen := s_osnovnoy_Wash;
			encoder_(reset := TRUE);
		ELSIF encoder_.counter >= 1 THEN
			encoder_(reset := TRUE);
		END_IF

	s_nastroyki:
		SelectScreen.str[1] := ' Температура    ';
		SelectScreen.str[2] := ' Время          ';
		SelectScreen.str[3] := ' Выход          ';


		SelectScreen(Qtyparam := 3, kbrd := kbrd);
		str := SelectScreen.str_out;
		encoder_(reset := TRUE);

		CASE SelectScreen.StrSelect OF
			0:	;
			1:	Current_screen     := s_tem;
			2:	Current_screen     := s_time;
			3:	Current_screen	   := s_osnovnoy_US_1;
		END_CASE

		IF SelectScreen.exit_scr THEN
			Current_screen := s_osnovnoy_US_1;
		END_IF

	s_tem:
		SelectScreen.str[1] := ' УЗВ1           ';
		SelectScreen.str[2] := ' УЗВ2           ';
		SelectScreen.str[3] := ' Ополаскивание  ';
		SelectScreen.str[4] := ' Сушка          ';
		SelectScreen.str[5] := ' Выход          ';

		SelectScreen(Qtyparam := 5, kbrd := kbrd);
		str := SelectScreen.str_out;

		CASE SelectScreen.StrSelect OF
			0:	;
			1:	Current_screen     := s_tem_us_1;
			2:	Current_screen     := s_tem_us_2;
			3:	Current_screen     := s_tem_wash;
			4:	Current_screen     := s_tem_dry;
			5:	Current_screen     := s_nastroyki;
		END_CASE

		IF SelectScreen.exit_scr THEN
			Current_screen := s_nastroyki;
		END_IF

	s_tem_us_1:
		SetScreen.str_in     := '  Температура УЗ';
		SetScreen.in_var_min := 1;
		SetScreen.in_var_max := tempMaxRet;
		SetScreen.UnitParam  := '$9BС';

		SetScreen.variable := BYTE_TO_VAR(APRet[US_1].byTemp);
		SetScreen(kbrd := kbrd, str_out => str);



		IF SetScreen.exit_screen THEN
			Current_screen := s_tem;
		END_IF

		IF SetScreen.next_screen THEN
			APRet[US_1].byTemp := DINT_TO_BYTE(SetScreen.ibuffer);
		END_IF

	s_tem_us_2:
		SetScreen.str_in     := '  Температура УЗ';
		SetScreen.in_var_min := 1;
		SetScreen.in_var_max := tempMaxRet;
		SetScreen.UnitParam  := '$9BС';

		SetScreen.variable := BYTE_TO_VAR(APRet[US_2].byTemp);
		SetScreen(kbrd := kbrd, str_out => str);



		IF SetScreen.exit_screen THEN
			Current_screen := s_tem;
		END_IF

		IF SetScreen.next_screen THEN
			APRet[US_2].byTemp := DINT_TO_BYTE(SetScreen.ibuffer);
		END_IF

	s_tem_wash:				  (*|   4   4   4   ||  4   4   4   |*)
		SetScreen.str_in     := '  Температура    ополаскивания  ';
		SetScreen.in_var_min := 1;
		SetScreen.in_var_max := tempMaxRet;
		SetScreen.UnitParam  := '$9BС';

		SetScreen.variable := BYTE_TO_VAR(APRet[Wash].byTemp);
		SetScreen(kbrd := kbrd, str_out => str);



		IF SetScreen.exit_screen THEN
			Current_screen := s_tem;
		END_IF

		IF SetScreen.next_screen THEN
			APRet[Wash].byTemp := DINT_TO_BYTE(SetScreen.ibuffer);
		END_IF


	s_tem_dry:				  (*|   4   4   4   ||  4   4   4   |*)
		SetScreen.str_in     := '  Температура        сушки      ';
		SetScreen.in_var_min := 1;
		SetScreen.in_var_max := 120;
		SetScreen.UnitParam  := '$9BС';

		SetScreen.variable := WORD_TO_VAR(temp_Air);
		SetScreen(kbrd := kbrd, str_out => str);



		IF SetScreen.exit_screen THEN
			Current_screen := s_tem;
		END_IF

		IF SetScreen.next_screen THEN
			temp_Air := DINT_TO_WORD(SetScreen.ibuffer);
		END_IF

	s_time:
		SelectScreen.str[1] := ' УЗВ1           ';
		SelectScreen.str[2] := ' УЗВ2           ';
		SelectScreen.str[3] := ' Сушка          ';
		SelectScreen.str[4] := ' Выход          ';

		SelectScreen(Qtyparam := 4, kbrd := kbrd);
		str := SelectScreen.str_out;
		encoder_(reset := TRUE);

		CASE SelectScreen.StrSelect OF
			0:	;
			1:	Current_screen     := s_time_us_1;
			2:	Current_screen     := s_time_us_2;
			3:	Current_screen     := s_time_dry;
			4:	Current_screen     := s_nastroyki;
		END_CASE

		IF SelectScreen.exit_scr THEN
			Current_screen := s_nastroyki;
		END_IF

	s_time_us_1:				  (*|   4   4   4   ||  4   4   4   |*)
		SetScreen.str_in     := '  Время работы    ультразвука   ';
		SetScreen.in_var_min := 0;
		SetScreen.in_var_max := timeMaxRet;
		SetScreen.UnitParam  := ' мин';

		SetScreen.variable := WORD_TO_VAR(APRet[US_1].arwTime[2]);
		SetScreen(kbrd := kbrd, str_out => str);

		IF SetScreen.exit_screen THEN
			Current_screen := s_time;
		END_IF

		IF SetScreen.next_screen THEN
			APRet[US_1].arwTime[2] := DINT_TO_WORD(SetScreen.ibuffer);
		END_IF

	s_time_us_2:				  (*|   4   4   4   ||  4   4   4   |*)
		SetScreen.str_in     := '  Время работы    ультразвука   ';
		SetScreen.in_var_min := 0;
		SetScreen.in_var_max := timeMaxRet;
		SetScreen.UnitParam  := ' мин';

		SetScreen.variable := WORD_TO_VAR(APRet[US_2].arwTime[2]);
		SetScreen(kbrd := kbrd, str_out => str);

		IF SetScreen.exit_screen THEN
			Current_screen := s_time;
		END_IF

		IF SetScreen.next_screen THEN
			APRet[US_2].arwTime[2] := DINT_TO_WORD(SetScreen.ibuffer);
		END_IF

	s_time_dry:				  (*|   4   4   4   ||  4   4   4   |*)
		SetScreen.str_in     := '  Время работы       сушки      ';
		SetScreen.in_var_min := 1;
		SetScreen.in_var_max := timeMaxRet;
		SetScreen.UnitParam  := ' мин';

		SetScreen.variable := WORD_TO_VAR(time_dry);
		SetScreen(kbrd := kbrd, str_out => str);

		IF SetScreen.exit_screen THEN
			Current_screen := s_time;
		END_IF

		IF SetScreen.next_screen THEN
			time_dry := DINT_TO_WORD(SetScreen.ibuffer);
		END_IF


	s_nastroyki_ext:
		SelectScreen.str[1] := ' Макс. темп.    ';
		SelectScreen.str[2] := ' Ширина гист.   ';

		SelectScreen(kbrd := kbrd, QtyParam := 2);
		str := SelectScreen.str_out;


		CASE SelectScreen.StrSelect OF
			0:	;
			1:	Current_screen := s_tMaxSet;
			2:	Current_screen := s_temHSet;
		END_CASE

		IF SelectScreen.exit_scr THEN
		Current_screen := s_osnovnoy_US_1;
		END_IF

	s_tMaxSet:
		SetScreen.str_in     := ' Максимальная   температура ';
		SetScreen.in_var_min := 1;
		SetScreen.in_var_max := 999;
		SetScreen.UnitParam  := '$9BС';

		SetScreen.variable := BYTE_TO_VAR(tempMaxRet);
		SetScreen(kbrd := kbrd, str_out => str);



		IF SetScreen.exit_screen THEN
			Current_screen := s_nastroyki_ext;
		END_IF

		IF SetScreen.next_screen THEN
			tempMaxRet := DINT_TO_BYTE(SetScreen.ibuffer);
		END_IF

	s_temHSet:
		SetScreen.str_in     := '     Ширина       гистерезиса   ';
		SetScreen.in_var_min := 2;
		SetScreen.in_var_max := 998;
		SetScreen.UnitParam  := '/10$9BС';

		SetScreen.variable := WORD_TO_VAR(hystRet);
		SetScreen(kbrd := kbrd, str_out => str);


		IF SetScreen.exit_screen THEN
			Current_screen := s_nastroyki_ext;
		END_IF

		IF SetScreen.next_screen THEN
			hystRet := DINT_TO_BYTE(SetScreen.ibuffer);
		END_IF

END_CASE


FOR I :=1 TO 4 BY 1 DO
	str[I]:=FillSpaceString(str[I],16);
	IF str[I]<>pred_str[I] THEN
		Write_Display(SINGLE_MODE,0,INT_TO_BYTE(I-1),str[I]);
		pred_str[I]:=str[I];
	END_IF
END_FOR
END_ACTION
ACTION acInit:
(*инициализация АП*)
bInit := APRet[US_1].areSt[2] = US;
IF NOT(bInit) THEN
	APRet[US_1].areSt[1]	:= WarmBath;
	APRet[US_1].byTemp		:= 60;
	APRet[US_1].areSt[2]	:= US;
	APRet[US_1].arwTime[2]	:= 1;

	APRet[US_2].areSt[1]	:= WarmBath;
	APRet[US_2].byTemp		:= 60;
	APRet[US_2].areSt[2]	:= US;
	APRet[US_2].arwTime[2]	:= 1;

	APRet[Wash].areSt[1]	:= WarmBath;
	APRet[Wash].byTemp		:= 30;

END_IF
FOR i := US_1 TO Wash DO
    block[i].pBath	      := ADR(bath[i]);
END_FOR
END_ACTION
ACTION acMB:
IF NOT(bOpenPort) THEN
	stSettings.byParity     := 0;
	stSettings.byStopBits   := 0;
	stSettings.dwBaudRate   := 9600;
	stSettings.dwBufferSize := 0;
	stSettings.dwScan       := 0;
	stSettings.dwTimeout    := 0;
	stSettings.Port         := ePorts;
	oComService(Enable:=NOT(bOpenPort),Settings:=stSettings,Task:=OPEN_TSK);
	IF oComService.Ready THEN
		bOpenPort := TRUE;
	END_IF
ELSE
	CASE eMBStep OF

		MV110Read:
			TONMBDelay(IN := NOT TONMBDelay.Q,PT := tMBDelay);
			IF TONMBDelay.Q THEN
			oMB_03(
				Enable    := TRUE,             (*разрешение работы блока*)
				Mode      := MB_RTU,           (*режим передачи*)
				DevAddr   := byMV110Address,    (*адрес*)
				FirstAddr := 51,                (*регистр битовая маска входов*)
				Quantity  := 1,                 (*количество регистров*)
				ComHandle := stSettings.Port,  (*настройки сом-порта*)
				TimeOut   := tTimeOut,          (*таймаут*)
				Buffer    := arMBuffer,         (*буфер данных*)
				);
			IF oMB_03.Complete AND oMB_03.Exception = 0 THEN
				udErr   := 0;
				eMBStep := MU110Write;
				wBuffer := BYTE_TO_WORD(arMBuffer[1])
				OR SHL(BYTE_TO_WORD(arMBuffer[0]), 8);
				mbA2    := wBuffer;
			END_IF
			IF oMB_03.Complete AND oMB_03.Exception <> 0 THEN
				eMBStep := MU110Write;
				udErr   := udErr + 1;
			END_IF
			END_IF
		MU110Write:
			TONMBDelay(IN := NOT TONMBDelay.Q,PT := tMBDelay);
			IF TONMBDelay.Q THEN
			IF NOT(oMB_16.Enable) THEN
				(* подготавливаем данные для отправки *)
				arMBuffer[0] := 0;
				arMBuffer[1] := 0;
				arMBuffer[1].0 := block[US_1].ContrOut.warmBath;
				arMBuffer[1].1 := block[US_2].ContrOut.warmBath;
				arMBuffer[1].2 := block[Wash].ContrOut.warmBath;
				arMBuffer[1].3 := contr.heat_air;
				arMBuffer[1].4 := TRUE;
				arMBuffer[1].5 := contr.fan;
				arMBuffer[1].6 := block[US_1].ContrOut.us;
				arMBuffer[1].7 := block[US_2].ContrOut.us;
			END_IF
			
			oMB_16(                            (*модбас функция 16*)
				Enable    := TRUE,             (*разрешение работы блока*)
				Mode      := MB_RTU,           (*режим передачи*)
				DevAddr   := byMU110Address,   (*адрес*)
				FirstAddr := 50,               (*регистр битовая маска входов*)
				Quantity  := 1,                (*количество регистров*)
				Buffer    := arMBuffer,        (*что передаем *)
				ComHandle := stSettings.Port,  (*номер сом-порта*)
				TimeOut   := tTimeOut,         (*таймаут*)
				);

			IF oMB_16.Complete THEN
				IF oMB_16.Exception = 0 THEN
					eMBStep := MV110Read;
					udErr   := 0;
				ELSE
					eMBStep := MV110Read;
					udErr   := udErr + 1;
				END_IF
				oMB_16(Enable := FALSE, Buffer := arMBuffer);
			END_IF
			END_IF
	END_CASE
END_IF
END_ACTION

(* POU FBv1/Encoder, ST *)
FUNCTION_BLOCK Encoder
VAR_INPUT
	A:            BOOL;
	B:            BOOL;
	button:       BOOL;
	reset:        BOOL;
	enable:       BOOL;
	connected:    BOOL := FALSE;
END_VAR
VAR_OUTPUT
	press:        BOOL;
	counter:      INT;
END_VAR
VAR
	AC:           BOOL;
END_VAR
IF A <> AC THEN
	IF B <> A THEN
		counter := counter + 1;
	ELSIF B = A THEN
		counter := counter - 1;
	END_IF
END_IF

AC       := A;
press    := button;

IF reset THEN
	counter := 0;
END_IF
END_FUNCTION_BLOCK

(* POU BFBv2/BFBv4, ST *)
FUNCTION_BLOCK BFBv4
VAR_INPUT
    stAP:               APST;            (*параметры автоматической программы*)
    sens:               SensorBath;      (*состояние датчиков*)
    Param:              ExtParamST;      (*дополнительные параметры*)
END_VAR
VAR_OUTPUT
    contr:              ControlBath;     (*управление*)
    extOutB:            ExtOutST;        (*дополнительные выходы ванны*)
    eStAP:              StAPE;
END_VAR
VAR
    bInit:              BOOL;            (*флаг инициализации*)
    iNSt:               INT     :=1;
    oHeatBath:          HYST;            (*ФБ нагрева ванны*)
	oHeatAir:			HYST;
	oHeatTank:          HYST;            (*ФБ нагрева бака*)
    TONStep:            TONP;            (*таймер состояния с паузой*)
    TONVent:            TON;             (*таймер открытия вентиля*)
    TONDelay:           TON;
    TONRot:             TON;             (*таймер периода качания*)
    TONRotDur:          TON;             (*таймер продолжительности качания*)
    TONRotSlack:        TON;             (*таймер бездействия качания*)
    BLINKMix:           BLINK;           (*блинкер перемешивания*)
    BLINKSkim:          BLINK;           (*блинкер скиммера*)
    filtrAvailable:     BOOL;            (*флаг доступности насоса*)
    barbAvailable:      BOOL;            (*флаг доступности барботажа*)
    autoAvailable:      BOOL;            (*флаг установки с гидролоками*)

    iSt:                INT;             (*переменная шага*)
    skimStart:          BOOL;            (*фиксация включения скиммера*)
    justBool:           BOOL;
    firstIntoFill:      BOOL    := TRUE; (*первый вход в заполнение*)
    TONAddFill:         TON;             (*таймер доп. налива*)
    addFill:            TIME    := t#3s; (*время до активации доп.налива*)

END_VAR
VAR_TEMP
    i:                  INT;
END_VAR
CASE eStAP OF
    Wait:
        IF Sens.button.Pusk THEN
            iNSt  := 1;
            eStAP := stAP.areSt[1];
        END_IF




    WarmBath:
        IF NOT(EXTRACT(stAP.byBool, WarmWait)) OR Sens.tempBath >= stAP.byTemp THEN
            acNextStep();
        END_IF
        acStop();

    US:
        Contr.us := stAP.arwTime[iNSt] <> 0;
        TONStep(P := Sens.pause, IN := TRUE,
        		PT := TO_MIN(stAP.arwTime[iNSt]));
        IF TONStep.Q THEN
            TONStep(IN := FALSE);
            Contr.us := FALSE;
            acNextStep();
        END_IF
        acStop();

    Barb:
        Contr.ventBarb := stAP.arwTime[iNSt] <> 0;
        TONStep(P := Sens.pause, IN := TRUE,
				PT := TO_MIN(stAP.arwTime[iNSt]));
        IF TONStep.Q THEN
            TONStep(IN := FALSE);
            Contr.ventBarb := FALSE;
            acNextStep();
        END_IF
        acStop();

END_CASE



(*нагрев*)
oHeatBath.temperatura := stAP.byTemp;
oHeatBath(ENABLE := Sens.warmOn, temInput := Sens.tempBath, temperaturaH := Param.deltaHyst);
Contr.warmBath := oHeatBath.nagrev;

(*Сушка*)
oHeatAir.temperatura := stAP.byTemp;
oHeatBath(ENABLE := Sens.warmOn, temInput := Sens.tempBath, temperaturaH := Param.deltaHyst);
Contr.warmBath := oHeatBath.nagrev;

(*расчет оставшегося времени шага*)
extOutB.remTime := TO_MIN(stAP.arwTime[iNSt]) - TONStep.ET;
END_FUNCTION_BLOCK
ACTION acNextStep:
iNSt  := iNSt + 1;
eStAP := stAP.areSt[iNSt];
IF eStAP = Wait OR iNSt = iStQty + 1 THEN
    iNSt := 1;
END_IF

firstIntoFill := TRUE;
TONAddFill(IN:=FALSE);
END_ACTION
ACTION acStop:
IF Sens.button.Stop OR sens.button.emStop THEN
    TONStep                 (IN:=FALSE);
    TONVent                 (IN:=FALSE);
    TONDelay                (IN:=FALSE);
    TONAddFill              (IN:=FALSE);
    eStAP                   := Wait;
    iNSt                    := 1;
    Contr.pumpBfromTank     := FALSE;
    Contr.rotFo             := FALSE;
    Contr.rotRe             := FALSE;
    Contr.us                := FALSE;
    Contr.ventBfromNet      := FALSE;
    Contr.ventBPocketToNet  := FALSE;
    Contr.ventBPocketToTank	:= FALSE;
    Contr.ventBToNet        := FALSE;
    Contr.ventBToTank       := FALSE;
    Contr.ventBarb          := FALSE;
    firstIntoFill           := TRUE;
END_IF
END_ACTION

(* POU FBv1/HYST, ST *)
FUNCTION_BLOCK HYST
VAR_INPUT
    enable:        BOOL    := TRUE;
    temInput:      REAL;
    temperatura:   DWORD;
    temperaturaH:  DWORD;
END_VAR
VAR_OUTPUT
    nagrev:        BOOL;
END_VAR
VAR

END_VAR
IF temInput<(DWORD_TO_REAL(temperatura)-(DWORD_TO_REAL(temperaturaH)/20)) THEN
    nagrev:=TRUE;
END_IF

IF temInput>(DWORD_TO_REAL(temperatura)+(DWORD_TO_REAL(temperaturaH)/20)) THEN
    nagrev:=FALSE;
END_IF


nagrev := nagrev AND enable;
END_FUNCTION_BLOCK

(* POU FBv1/TONP, ST *)
(*блок таймера с паузой*)
FUNCTION_BLOCK TONP
VAR_INPUT
    P:     BOOL;    (*Пауза*)
    IN:    BOOL;
    PT:    TIME;
END_VAR
VAR_OUTPUT
    Q:     BOOL;
    ET:    TIME;
END_VAR
VAR
    TON1:  TON;
    t:     TIME;
END_VAR
IF P THEN
    t  := MAX(TON1.ET + t, t);
    ET := t;
ELSE
    ET := TON1.ET + t;
END_IF
TON1(IN := IN AND NOT(P), PT := PT - t);
Q := TON1.Q;
IF (*Q AND*) NOT(IN) THEN
    t := t#0m0s0ms;
    P := FALSE;
END_IF
END_FUNCTION_BLOCK

(* POU FUNv1/TO_MIN, ST *)
FUNCTION TO_MIN : TIME
VAR_INPUT
	in: DWORD;
END_VAR
VAR
END_VAR
TO_MIN := DWORD_TO_TIME(in)*60000;
END_FUNCTION

(* POU BFBv2/BlockFBv2, ST *)
FUNCTION_BLOCK BlockFBv2
VAR_INPUT
    pBath:             POINTER TO BFBv4;
END_VAR
VAR_OUTPUT
    ContrOut:          ControlBath;
   (*оставшееся время задержки повторного включения УЗ*)
    tUSDelayRemain:    TIME;
END_VAR
VAR
    (*таймер блокировки от многократного включения УЗ*)
    TONUSBl:           TON;
    bUSwasOn:          BOOL;
END_VAR
ContrOut:=pBath^.Contr;

(*Блокировка ТЭН в ванне или баке*)
IF pBath^.Param.heaterInTank THEN
    ContrOut.warmBath := pBath^.Contr.warmBath
    AND pBath^.Sens.level.WarmBlock AND pBath^.Sens.tempBath>0;
ELSE
    ContrOut.warmBath := pBath^.Contr.warmBath
                     AND pBath^.Sens.level.WarmBlock
                     AND pBath^.Sens.tempBath>0;
END_IF


(*Блокирковка насоса*)
ContrOut.pumpBfromTank := pBath^.contr.pumpBfromTank
						AND pBath^.sens.level.PumpBlock
						AND NOT (pBath^.sens.pause)
						AND pBath^.sens.overloadPump;


(*Блокировка ультразвука*)
ContrOut.us := pBath^.contr.us
           AND pBath^.sens.level.USBlock
           AND NOT(pBath^.sens.pause)
           AND NOT(TONUSBl.IN);
IF bUSwasOn > ContrOut.us THEN
    TONUSBl.IN     := TRUE;
    tUSDelayRemain := WORD_TO_TIME(USDelayRet) * 1000 - TONUSBl.ET;
ELSE
	tUSDelayRemain := t#0ms;
END_IF
TONUSBl(PT:=WORD_TO_TIME(USDelayRet) * 1000);
IF NOT(TONUSBl.IN) OR  TONUSBl.Q THEN
    TONUSBl.IN := FALSE;
    bUSwasOn   := ContrOut.us;
END_IF

(*Блокировка барботажа*)
ContrOut.ventBarb:=pBath^.Contr.ventBarb AND pBath^.Sens.level.BarbBlock;
END_FUNCTION_BLOCK

(* POU FBv1/digitalFiltr, ST *)
FUNCTION_BLOCK digitalFiltr
VAR_INPUT
    In:     BOOL;
END_VAR
VAR_OUTPUT
    Out:    BOOL;
END_VAR
VAR
    TON_:   TON;
END_VAR
TON_(IN:=In<>Out,PT:=(DWORD_TO_TIME(wFilterTimeRet)));
IF TON_.Q THEN
    TON_(IN:=FALSE);
    Out:=In;
END_IF
END_FUNCTION_BLOCK

(* POU FBv1/KeyboardFB, ST *)
(*блок клавиатура*)
FUNCTION_BLOCK KeyboardFB
VAR_IN_OUT
    kbrd:         WORD;
END_VAR
VAR_INPUT
END_VAR
VAR_OUTPUT
    OFF:          BOOL;
    DOWN:         ButtonEvent;
    UP:           ButtonEvent;
    ENTER:        ButtonEvent;
    OUT:          ButtonEvent;
    ALT:          ButtonEvent;
    F1:           ButtonEvent;
    F2:           ButtonEvent;
    F3:           ButtonEvent;
    PUSK_STOP:    ButtonEvent;
    ALT_F1:       ButtonEvent;
    ALT_F3:       ButtonEvent;
END_VAR
VAR
    iSt:          INT;
	(* указатель на устанавливемый/снимаемый сигнал *)
    pBut:         POINTER TO ButtonEvent;
    kbrdLastTime: WORD;
    TON_:         TON;
    TONincr:      TON;
    lastIncr:     BYTE;
END_VAR
VAR_TEMP

END_VAR
CASE iSt OF
    0:	(* init *)
        pBut     := ADR(ALT);
        TON_(IN:= FALSE, PT := t#1s);
        lastIncr := 1;
        iSt      := 1;

    1:	(* down *)
        pBut^.downEvent := FALSE;
        pBut^.incr := 0;
        IF kbrd <> 0 AND kbrd <> kbrdLastTime THEN
            acSetPointerToBool();
            pBut^.downEvent := TRUE;
            pBut^.incr      := 1;
        END_IF
        TON_(IN:= kbrd<>0, PT := t#1s);
        IF TON_.Q THEN
            TON_(IN := FALSE);
            pBut^.longPush := TRUE;
            pBut^.incr     := 1;
            iSt            := 2;
        END_IF

    2:	(* longPush *)
        pBut^.incr := 0;
        TON_(IN := TRUE, PT := t#200ms);
        IF TON_.Q THEN
            TON_(IN:=FALSE);
            pBut^.incr := lastIncr;
        END_IF
        TONincr(IN := TRUE, PT := t#1s);
        IF TONincr.Q THEN
            TONincr(IN := FALSE);
            lastIncr := lastIncr + 1;
        END_IF
        IF kbrd = 0 OR kbrd <> kbrdLastTime THEN
            pBut^.longPush := FALSE;
            TON_(IN := FALSE);
            pBut^.incr     := 0;
            lastIncr       := 1;
            iSt            := 1;
        END_IF

END_CASE
kbrdLastTime := kbrd;
OFF          := kbrd = 0;
END_FUNCTION_BLOCK
ACTION acSetPointerToBool:
CASE kbrd OF
    1:      pBut := ADR(F1);
    2:      pBut := ADR(F2);
    4:      pBut := ADR(DOWN);
    8:      pBut := ADR(UP);
    16:     pBut := ADR(ENTER);
    32:     pBut := ADR(PUSK_STOP);
    64:     pBut := ADR(OUT);
    128:    pBut := ADR(ALT);
    256:    pBut := ADR(F3);
    129:    pBut := ADR(ALT_F1);
    384:    pBut := ADR(ALT_F3);
END_CASE
END_ACTION

(* POU FBv1/SelectScreenFB, ST *)
(*блок экрана выбора параметров кареткой (до iMaxSelScrParam)*)
FUNCTION_BLOCK SelectScreenFB
VAR_INPUT
    (*строки с кратким описание параметров*)
    str:         ARRAY [1..iMaxSelScrParam] OF STRING(16);
    (*количество параметров*)
    QtyParam:    INT;
    (*клавиатура управления*)
    kbrd:        kbrd_tip;
    (*расширенная структура для дописывания в свободное место 4-й строки*)
    ext:         SelectScreenAddStruc;
	pressLastTime: BOOL;
	encoder_:       Encoder;
END_VAR
VAR_OUTPUT
    str_out:     ARRAY [1..4] OF STRING(16);
    StrSelect:   UINT;
END_VAR
VAR
    karetka:     UINT    :=1;
    action_done: BOOL;
    FirstIn:     BOOL    :=TRUE;
    exit_scr:    BOOL;
	TON_:        TON;
END_VAR
VAR_TEMP
    (*номер параметра из str в каждой строке экрана, параметр, равный 0 - пустая строка*)
    N:           ARRAY [1..3] OF INT:=3(0);
    i:           INT;
END_VAR
StrSelect := 0;StrSelect := 0;
exit_scr  := FALSE;
FOR i := 1 TO 3 DO
    N[i] := 0;
END_FOR
IF FirstIn AND (kbrd <> OFF OR encoder_.press AND encoder_.connected) THEN
    action_done   := TRUE;
ELSE
    FirstIn := FALSE;
END_IF


(*определение положения каретки и параметра каждй строки*)
IF karetka = 1 THEN
    FOR i := 1 TO MIN(QtyParam, 3) DO
        N[i] := i;
        str_out[i] := SEL(i = 1, ' ', '$B0');
    END_FOR
(*	str_out[1]:='$B0'; str_out[2]:=' '; str_out[3]:=' ';*)
ELSIF karetka = QtyParam THEN
    FOR i := MIN(QtyParam, 3) TO 1 BY -1 DO
        N[i] := QtyParam + i - MIN(QtyParam, 3);
        str_out[i] := SEL(i = MIN(QtyParam, 3), ' ', '$B0');
    END_FOR
(*	str_out[1]:=' '; str_out[2]:=' '; str_out[3]:='$B0';*)
ELSE
    N[1] := karetka - 1; N[2] := karetka; N[3] := karetka + 1;
    str_out[1] := ' '; str_out[2] := '$B0'; str_out[3] := ' ';
END_IF
IF karetka > 2 THEN
    str_out[1] := '$A1';
END_IF
IF karetka < QtyParam - 1 THEN
    str_out[3] := '$A2';
END_IF
karetka := SEL(karetka > QtyParam, karetka, QtyParam);


FOR i := 1 TO 3 DO
    str_out[i] := SEL(N[i] = 0,	CONCAT(str_out[i], LEFT(str[N[i]], 15)), '');
    (*	IF (*LEN(str[N[i]])<=15 AND*) N[i]<>0  THEN
    str_out[i]:=CONCAT(str_out[i],LEFT(str[N[i]],15);
    ELSE
    str_out[i]:='';
    END_IF
    *)
END_FOR

IF LEN(ext.strIn) = 1 THEN
    str_out[4] := CONCAT('ВЫХОД   ', ext.strIn);
    str_out[4] := CONCAT(str_out[4], '   ВВОД');
ELSIF LEN(ext.strIn) = 2 THEN
    str_out[4] := CONCAT('ВЫХОД  ', ext.strIn);
    str_out[4] := CONCAT(str_out[4], '   ВВОД');
ELSIF LEN(ext.strIn) = 3 THEN
    str_out[4] := CONCAT('ВЫХОД  ', ext.strIn);
    str_out[4] := CONCAT(str_out[4], '  ВВОД');
ELSIF LEN(ext.strIn) = 4 THEN
    str_out[4] := CONCAT('ВЫХОД ', ext.strIn);
    str_out[4] := CONCAT(str_out[4], '  ВВОД');
ELSIF LEN(ext.strIn) = 5 THEN
    str_out[4] := CONCAT('ВЫХОД ', ext.strIn);
    str_out[4] := CONCAT(str_out[4], ' ВВОД');
ELSE
    str_out[4] := 'ВЫХОД       ВВОД';
END_IF

IF NOT(action_done) AND kbrd <> OFF THEN
    action_done := TRUE;
    CASE kbrd OF
        UP:     karetka   := MAX(karetka - 1, 1);
        DOWN:   karetka   := MIN(karetka + 1, QtyParam);
        ENTER:  StrSelect := karetka; FirstIn  := TRUE;
        OUT:    FirstIn   :=TRUE;     exit_scr := TRUE;
    END_CASE
END_IF

IF encoder_.connected THEN
	IF NOT(action_done) AND encoder_.connected THEN
	    action_done := TRUE;
		acENC();
		encoder_(reset := FALSE);
	END_IF


	IF encoder_.enable THEN
		IF encoder_.press <> pressLastTime AND NOT (encoder_.press OR TON_.Q) THEN
			action_done := TRUE;
			encoder_(enable := FALSE);
			StrSelect := karetka; FirstIn  := TRUE;
		END_IF
		TON_(IN:= encoder_.press <> 0, PT := t#1s);
		IF TON_.Q THEN
			TON_(IN := FALSE);
			action_done := TRUE;
			encoder_(enable := FALSE);
			FirstIn   :=TRUE;     exit_scr := TRUE;
		END_IF
	END_IF
	pressLastTime := encoder_.press;
END_IF

IF NOT encoder_.press THEN
	encoder_(enable := TRUE);
END_IF
IF kbrd = OFF THEN
    action_done := FALSE;
END_IF
END_FUNCTION_BLOCK
ACTION acENC:
IF ((karetka + encoder_.counter) > 1) AND ((karetka + encoder_.counter) < QtyParam) THEN
	karetka := karetka + encoder_.counter;
	encoder_(reset := TRUE);
ELSIF (karetka + encoder_.counter) <= 1 THEN
	karetka := 1;
	encoder_(reset := TRUE);
ELSIF (karetka + encoder_.counter) >= QtyParam THEN
	karetka := QtyParam;
	encoder_(reset := TRUE);
END_IF
END_ACTION

(* POU FBv1/SetScreenFB, ST *)
(*блок экрана задания параметров*)
FUNCTION_BLOCK SetScreenFB
VAR_INPUT
    (*мин значение задаваемой переменной*)
    in_var_min:     DINT;
    (*макс значение задаваемой переменной*)
    in_var_max:     DINT;
    (*мин значение задаваемой переменной*)
    in_var_min_r:   REAL;
    (*макс значение задаваемой переменной*)
    in_var_max_r:   REAL;

    (*в каких единицах ведется задание минуты секунды градусы и тд*)
    UnitParam:      STRING;
    (*клавиатура ПЛК73*)
    kbrd:           kbrd_tip;

    (*текстовое описание переменной строки 1,2 вместе (обязательно 32 символа)*)
    str_in:         STRING(32);

    (*указательна изменяемый параметр*)
    pby:            POINTER TO BYTE;
    (*размер изменяемого параметра*)
    bySize:         INT;
    variable:       VarST;
    ibufferD:       DINT;
    ibufferOst:     DINT;
	pSelect:        POINTER TO SelectScreenFB;
	encOut:         INT;
    enc:            DINT;
    enc_r:          REAL;
END_VAR

VAR_OUTPUT
    (*массив выводимых на экран строк*)
    str_out:        ARRAY [1..4] OF STRING(16);
    (*измененное значение переменной*)
    out_varExt:     ARRAY [1..3] OF DWORD;
    (*переменная выхода из экрана*)
    exit_screen:    BOOL;
    (*переменная перехода к следующему экрану*)
    next_screen:    BOOL;


END_VAR
VAR
    step:           INT;
    ibuffer:        DINT;
    rbuffer:        REAL;
    bufferExt:      ARRAY[1..3] OF DWORD;
    UnitSel:        UINT               :=1;
    action_done:    BOOL;
    TON_kbrd:       TON;
    just_bool:      BOOL;
    FirstIn:        BOOL               :=TRUE;
    pw:             POINTER TO WORD;
    pdw:            POINTER TO DWORD;
    pr:             POINTER TO REAL;
    pdi:            POINTER TO DINT;
	pressLastTime:  BOOL;
	TON_:           TON;
END_VAR
exit_screen := FALSE;
next_screen := FALSE;
IF FirstIn AND (kbrd <> OFF OR pSelect^.encoder_.press AND pSelect^.encoder_.connected) THEN
    action_done := TRUE;
ELSE
    FirstIn := FALSE;
END_IF

str_in := FillSpaceString(str_in, 32);
str_out[1] := LEFT(str_in, 16);
str_out[2] := RIGHT(str_in, 16);
str_out[3] := '$A2/$A1 ';
CASE step OF
	0:
    	CASE variable.type_ OF
    		BYTE_:     ibuffer := variable.pby^;
    		WORD_:     pw  := variable.pby;     ibuffer:=pw^;
    		DWORD_:    pdw := variable.pby;     ibuffer:=pdw^;
    		REAL_:     pr  := variable.pby;     rbuffer:=pr^;
    		DINT_:     pdi := variable.pby;     ibuffer:=pdi^;
    		DWORD_30:  pdw := variable.pby;     ibuffer:=pdw^;
    		DWORD_500: pdw := variable.pby;     ibuffer:=pdw^;
    	END_CASE
        step := step + 1;
    1:	IF NOT(action_done) AND kbrd <> OFF THEN
			action_done := TRUE;
			CASE kbrd OF
				OUT:	exit_screen := TRUE; step := 0; FirstIn := TRUE;
				UP:		acUp();
				DOWN:	acDown();
				ENTER:	CASE variable.type_ OF
							BYTE_:     variable.pby^:=DINT_TO_BYTE(ibuffer);
							WORD_:     pw^  := DINT_TO_WORD(ibuffer);
							DWORD_:    pdw^ := DINT_TO_DWORD(ibuffer);
							REAL_:     pr^  := rbuffer;
							DINT_:     pdi^ := ibuffer;
							DWORD_30:  pdw^ := DINT_TO_DWORD(ibuffer);
							DWORD_500: pdw^ := DINT_TO_DWORD(ibuffer);
						END_CASE
				exit_screen := TRUE; step := 0; FirstIn := TRUE;
				next_screen:=TRUE;
			END_CASE
		END_IF
		IF pSelect^.encoder_.connected THEN
			IF NOT(action_done) THEN
				action_done := TRUE;
				acENC();
				pSelect^.encoder_(reset := FALSE);
			END_IF
	
	
			IF pSelect^.encoder_.enable THEN
				IF pSelect^.encoder_.press <> pressLastTime
					AND NOT (pSelect^.encoder_.press OR TON_.Q) THEN
					pSelect^.encoder_.enable := FALSE;
					action_done := TRUE;
					CASE variable.type_ OF
			            BYTE_:     variable.pby^:=DINT_TO_BYTE(ibuffer);
			            WORD_:     pw^  := DINT_TO_WORD(ibuffer);
			            DWORD_:    pdw^ := DINT_TO_DWORD(ibuffer);
			            REAL_:     pr^  := rbuffer;
			            DINT_:     pdi^ := ibuffer;
			            DWORD_30:  pdw^ := DINT_TO_DWORD(ibuffer);
			            DWORD_500: pdw^ := DINT_TO_DWORD(ibuffer);
		            END_CASE
					exit_screen := TRUE; step := 0; FirstIn := TRUE;
			        next_screen:=TRUE;
				END_IF
				TON_(IN:= pSelect^.encoder_.press <> 0, PT := t#1s);
				IF TON_.Q THEN
					TON_(IN := FALSE);
					action_done := TRUE;
					pSelect^.encoder_.enable := FALSE;
					exit_screen := TRUE; step := 0; FirstIn := TRUE;
				END_IF
			END_IF
			pressLastTime := pSelect^.encoder_.press AND NOT exit_screen;
		END_IF
		TON_kbrd(IN:=kbrd<>OFF, PT:=t#1s);
		IF TON_kbrd.Q THEN
			IF just_bool THEN
				CASE kbrd OF
					UP:		acUp();
					DOWN:	acDown();
				END_CASE
			END_IF
			just_bool := NOT(just_bool);
		END_IF
END_CASE

CASE variable.type_ OF
    REAL_:
        IF rbuffer < 10 AND rbuffer > -10 THEN
            str_out[3] := CONCAT(str_out[3], '  ');
        ELSIF rbuffer < 100 AND rbuffer > -100 THEN
            str_out[3] := CONCAT(str_out[3], ' ');
        END_IF
        str_out[3] := CONCAT(str_out[3], REAL_TO_STRING(rbuffer));
    DWORD_30:
        IF ibuffer < 10  THEN
            str_out[3] := CONCAT(str_out[3], '  ');
        ELSIF ibuffer < 600  THEN
            str_out[3] := CONCAT(str_out[3], ' ');
        END_IF
        ibufferD   := ibuffer / 60;
        ibufferOst := ibuffer / 6 MOD 10;
        str_out[3] := CONCAT(str_out[3], DINT_TO_STRING (ibufferD));
        str_out[3] := CONCAT(str_out[3], ',');
        str_out[3] := CONCAT(str_out[3], DINT_TO_STRING (ibufferOst));
    DWORD_500:
        IF ibuffer < 1000  THEN
            str_out[3] := CONCAT(str_out[3], '  ');
        ELSIF ibuffer < 10000  THEN
            str_out[3] := CONCAT(str_out[3], ' ');
        END_IF
    ibufferD := ibuffer / 1000;
    ibufferOst := ibuffer MOD 1000;
    str_out[3] := CONCAT(str_out[3], DINT_TO_STRING (ibufferD));
    str_out[3] := CONCAT(str_out[3], ',');
    str_out[3] := CONCAT(str_out[3], DINT_TO_STRING(ibufferOst));
ELSE
    IF ibuffer < 10 AND ibuffer > -10 THEN
        str_out[3] := CONCAT(str_out[3], '  ');
    ELSIF ibuffer < 100 AND ibuffer > -100 THEN
    str_out[3] := CONCAT(str_out[3], ' ');
    END_IF
    str_out[3] := CONCAT(str_out[3], DINT_TO_STRING(ibuffer));
END_CASE

str_out[3] := CONCAT(str_out[3], UnitParam);

str_out[4] := 'ВЫХОД       ВВОД';


IF kbrd = OFF  THEN
    action_done := FALSE;
END_IF

IF NOT pSelect^.encoder_.press THEN
	pSelect^.encoder_(enable := TRUE);
END_IF
END_FUNCTION_BLOCK
ACTION acDown:
CASE variable.type_ OF
    BYTE_:      ibuffer := MAX(ibuffer - 1, in_var_min);
    WORD_:      ibuffer := MAX(ibuffer - 1, in_var_min);
    DWORD_:     ibuffer := MAX(ibuffer - 1, in_var_min);
    REAL_:      rbuffer := MAX(rbuffer * 0.9, in_var_min);
    DINT_:      ibuffer := MAX(ibuffer - 1, in_var_min);
    DWORD_30:   ibuffer := MAX(ibuffer - 30, in_var_min);
    DWORD_500:  ibuffer := MAX(ibuffer - 500, in_var_min);
END_CASE
END_ACTION
ACTION acENC:
IF ((ibuffer + pSelect^.encoder_.counter) > in_var_min) AND ((ibuffer + pSelect^.encoder_.counter) < in_var_max) THEN
	CASE variable.type_ OF
	    BYTE_:      ibuffer := ibuffer + pSelect^.encoder_.counter;
	    WORD_:      ibuffer := ibuffer + pSelect^.encoder_.counter;
	    DWORD_:     ibuffer := ibuffer + pSelect^.encoder_.counter;
	    REAL_:      rbuffer := rbuffer + pSelect^.encoder_.counter;
	    DINT_:      ibuffer := ibuffer + pSelect^.encoder_.counter;
	    DWORD_30:   ibuffer := ibuffer + pSelect^.encoder_.counter * 30;
	    DWORD_500:  ibuffer := ibuffer + pSelect^.encoder_.counter * 500;
	END_CASE
	pSelect^.encoder_(reset := TRUE);
ELSIF (ibuffer + pSelect^.encoder_.counter) <= in_var_min THEN
	CASE variable.type_ OF
	    BYTE_:      ibuffer := in_var_min;
	    WORD_:      ibuffer := in_var_min;
	    DWORD_:     ibuffer := in_var_min;
	    REAL_:      rbuffer := in_var_min;
	    DINT_:      ibuffer := in_var_min;
	    DWORD_30:   ibuffer := in_var_min;
	    DWORD_500:  ibuffer := in_var_min;
	END_CASE
	pSelect^.encoder_(reset := TRUE);
ELSIF (ibuffer + pSelect^.encoder_.counter) >= in_var_max THEN
	CASE variable.type_ OF
	    BYTE_:      ibuffer := in_var_max;
	    WORD_:      ibuffer := in_var_max;
	    DWORD_:     ibuffer := in_var_max;
	    REAL_:      rbuffer := in_var_max;
	    DINT_:      ibuffer := in_var_max;
	    DWORD_30:   ibuffer := in_var_max;
	    DWORD_500:  ibuffer := in_var_max;
	END_CASE
	pSelect^.encoder_(reset := TRUE);
END_IF
END_ACTION
ACTION acUp:
CASE variable.type_ OF
    BYTE_:     ibuffer := MIN(ibuffer + 1, in_var_max);
    WORD_:     ibuffer := MIN(ibuffer + 1, in_var_max);
    DWORD_:    ibuffer := MIN(ibuffer + 1, in_var_max);
    DINT_:     ibuffer := MIN(ibuffer + 1, in_var_max);
    REAL_:     rbuffer := MIN(rbuffer * 1.1, in_var_max);
    DWORD_30:  ibuffer := MIN(ibuffer + 30, in_var_max);
    DWORD_500: ibuffer := MIN(ibuffer + 500, in_var_max);
END_CASE
END_ACTION

(* POU FUNv1/FillSpaceString, ST *)
(*заполняет строку пробелами до указанной длины*)
FUNCTION FillSpaceString : STRING
VAR_INPUT
    str:   STRING;
    index: UINT;
END_VAR
VAR
    i:     INT;
    ii:    INT;
END_VAR
ii := LEN(str);
FillSpaceString := str;
FOR i := ii TO index - 1 DO
    FillSpaceString := CONCAT(FillSpaceString, ' ');
END_FOR
END_FUNCTION

(* POU FUNv1/TIME_TO_MMSS, ST *)
FUNCTION TIME_TO_MMSS : STRING
VAR_INPUT
    t:       TIME;
END_VAR
VAR
    minuta:  DWORD;
    secunda: DWORD;
END_VAR
TIME_TO_MMSS := ':';
minuta       := TIME_TO_DWORD(t) / 60000;
secunda      := TIME_TO_DWORD(t) / 1000 MOD 60;
TIME_TO_MMSS := INSERT(TIME_TO_MMSS, DWORD_TO_STRING(minuta), 0);
IF minuta < 100 THEN
    TIME_TO_MMSS := CONCAT(' ', TIME_TO_MMSS);
END_IF
IF minuta < 10 THEN
    TIME_TO_MMSS := CONCAT(' ', TIME_TO_MMSS);
END_IF
IF secunda < 10 THEN
    TIME_TO_MMSS := CONCAT(TIME_TO_MMSS, '0');
END_IF;
TIME_TO_MMSS := CONCAT(TIME_TO_MMSS, DWORD_TO_STRING(secunda));
END_FUNCTION

(* POU FUNv1/TEMP_TO_STRING, ST *)
FUNCTION TEMP_TO_STRING : STRING
VAR_INPUT
	in:      REAL;
END_VAR
VAR
	temD:    INT;
	temOst:  INT;
END_VAR
temD := (REAL_TO_INT (in*10));
temOst := temD MOD 10;
temD := temD / 10;

IF temD < 10 THEN
TEMP_TO_STRING := (' ');
END_IF

TEMP_TO_STRING := CONCAT(INT_TO_STRING (temD),',');

TEMP_TO_STRING := CONCAT(TEMP_TO_STRING, INT_TO_STRING(temOst));
END_FUNCTION

(* POU FUNv1/BYTE_TO_VAR, ST *)
FUNCTION BYTE_TO_VAR : VarST
VAR_IN_OUT
    in: BYTE;
END_VAR
VAR
END_VAR
BYTE_TO_VAR.pby   := ADR(in);
BYTE_TO_VAR.type_ := BYTE_;
END_FUNCTION

(* POU FUNv1/WORD_TO_VAR, ST *)
FUNCTION WORD_TO_VAR : VarST
VAR_IN_OUT
    in : WORD;
END_VAR
VAR
END_VAR
WORD_TO_VAR.pby   := ADR(in);
WORD_TO_VAR.type_ := WORD_;
END_FUNCTION

(* POU FUNv1/TO_SEC, ST *)
FUNCTION TO_SEC : TIME
VAR_INPUT
	in: DWORD;
END_VAR
VAR
END_VAR
TO_SEC := DWORD_TO_TIME(in)*1000;
END_FUNCTION

